% RSLogix 500 project HOT_WATER_SUPPLY.RSS, saved by version 8.30.00.16 %
PROJECT "BRAIN_1"    % processor: Bul.1763 MicroLogix 1100 Series B %

PROGRAM FILES
  LAD 2 "MAIN"  10 rungs
  LAD 3 "DIGI IN"  9 rungs  % Digital Inputs %
  LAD 4 "DIGI OUT"  6 rungs  % Digital Output %
  LAD 5 "ANG IN"  3 rungs  % Analog Inputs %
  LAD 6 "ANG OUT"  2 rungs  % Analog Output %
  LAD 7 "CONTROLS"  13 rungs  % Hand, Off, Auto Modes %
  LAD 9 "ALARMS"  21 rungs  % Alarms & Notification Control %
  LAD 10 "DISPLAY"  2 rungs

DATA FILES
  O0 OUTPUT  6 elements
  I1 INPUT  18 elements
  S2 STATUS  66 elements
  B3 BINARY  6 elements
  T4 TIMER  9 elements
  C5 COUNTER  1 elements
  R6 CONTROL  1 elements
  N7 INTEGER  10 elements
  F8 FLOAT  2 elements
  PD9 PID  1 elements

LADDER 2 "MAIN"
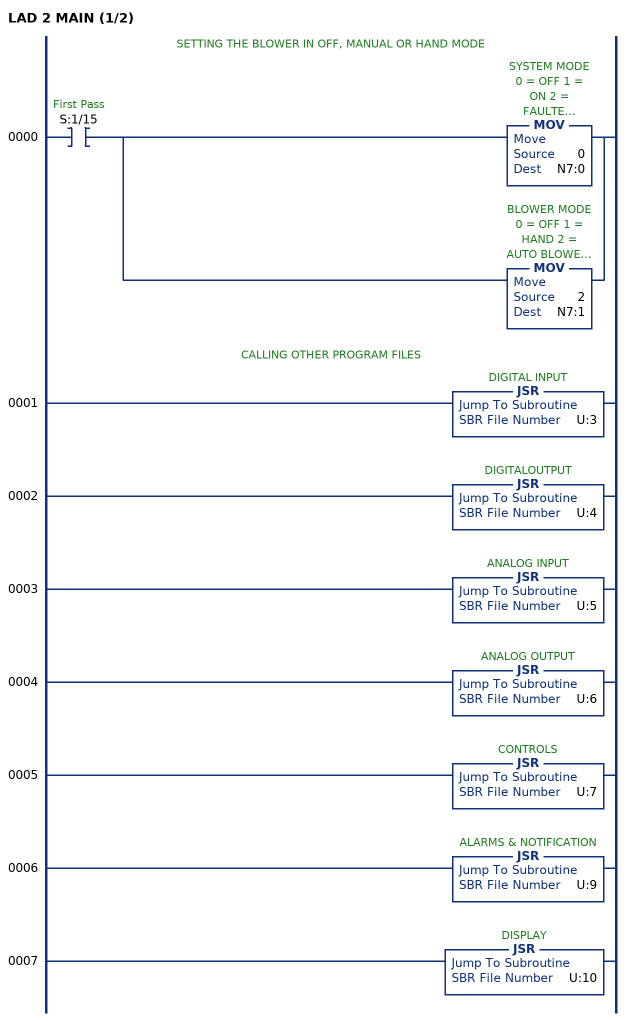
% Rung: 0 %
% SETTING THE BLOWER IN OFF, MANUAL OR HAND MODE %
SOR XIC S:1/15 BST MOV 0 N7:0 NXB MOV 2 N7:1 BND EOR
%   S:1/15  "First Pass" %
%   N7:0  SYSTEM_MODE  "SYSTEM MODE 0 = OFF 1 = ON 2 = FAULTED" %
%   N7:1  BLOWER_MODE  "BLOWER MODE 0 = OFF 1 = HAND 2 = AUTO" %
% Rung: 1 %
% CALLING OTHER PROGRAM FILES %
SOR JSR U:3 EOR
%   U:3  "DIGITAL INPUT" %
% Rung: 2 %
SOR JSR U:4 EOR
%   U:4  "DIGITALOUTPUT" %
% Rung: 3 %
SOR JSR U:5 EOR
%   U:5  "ANALOG INPUT" %
% Rung: 4 %
SOR JSR U:6 EOR
%   U:6  "ANALOG OUTPUT" %
% Rung: 5 %
SOR JSR U:7 EOR
%   U:7  "CONTROLS" %
% Rung: 6 %
SOR JSR U:9 EOR
%   U:9  "ALARMS & NOTIFICATION" %
% Rung: 7 %
SOR JSR U:10 EOR
%   U:10  "DISPLAY" %

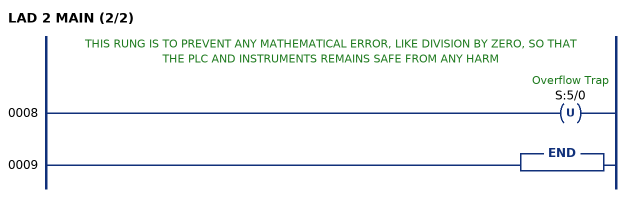
% Rung: 8 %
% THIS RUNG IS TO PREVENT ANY MATHEMATICAL ERROR, LIKE DIVISION BY ZERO, SO THAT THE PLC AND INSTRUMENTS REMAINS SAFE FROM ANY HARM %
SOR OTU S:5/0 EOR
%   S:5/0  "Overflow Trap" %
% Rung: 9 %
SOR END EOR

LADDER 3 "DIGI IN"    % Digital Inputs %
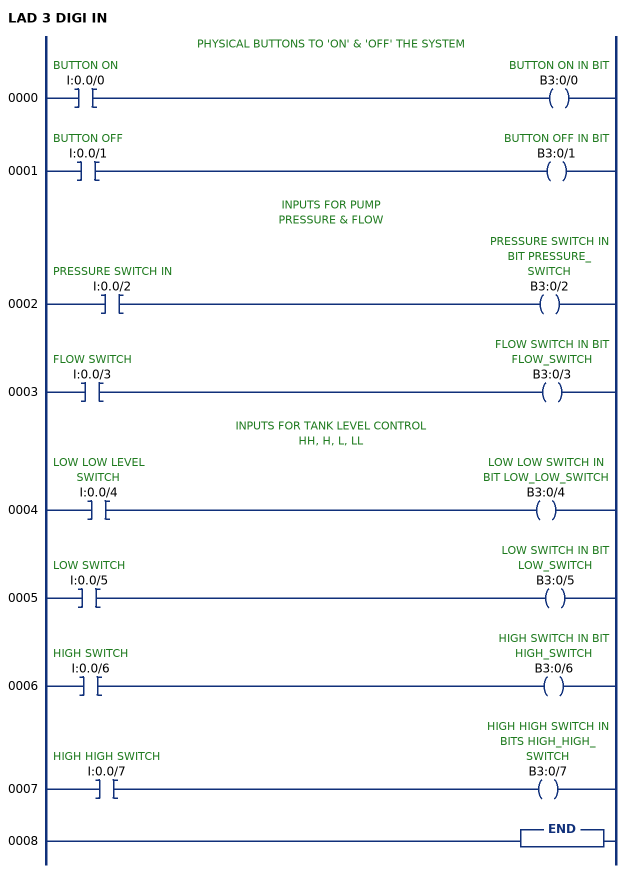
% Rung: 0 %
% PHYSICAL BUTTONS TO 'ON' & 'OFF' THE SYSTEM %
SOR XIC I:0.0/0 OTE B3:0/0 EOR
%   I:0.0/0  "BUTTON ON" %
%   B3:0/0  "BUTTON ON IN BIT" %
% Rung: 1 %
SOR XIC I:0.0/1 OTE B3:0/1 EOR
%   I:0.0/1  "BUTTON OFF" %
%   B3:0/1  "BUTTON OFF IN BIT" %
% Rung: 2 %
% INPUTS FOR PUMP
% PRESSURE & FLOW %
SOR XIC I:0.0/2 OTE B3:0/2 EOR
%   I:0.0/2  "PRESSURE SWITCH IN" %
%   B3:0/2  PRESSURE_SWITCH  "PRESSURE SWITCH IN BIT" %
% Rung: 3 %
SOR XIC I:0.0/3 OTE B3:0/3 EOR
%   I:0.0/3  "FLOW SWITCH" %
%   B3:0/3  FLOW_SWITCH  "FLOW SWITCH IN BIT" %
% Rung: 4 %
% INPUTS FOR TANK LEVEL CONTROL
% HH, H, L, LL %
SOR XIC I:0.0/4 OTE B3:0/4 EOR
%   I:0.0/4  "LOW LOW LEVEL SWITCH" %
%   B3:0/4  LOW_LOW_SWITCH  "LOW LOW SWITCH IN BIT" %
% Rung: 5 %
SOR XIC I:0.0/5 OTE B3:0/5 EOR
%   I:0.0/5  "LOW SWITCH" %
%   B3:0/5  LOW_SWITCH  "LOW SWITCH IN BIT" %
% Rung: 6 %
SOR XIC I:0.0/6 OTE B3:0/6 EOR
%   I:0.0/6  "HIGH SWITCH" %
%   B3:0/6  HIGH_SWITCH  "HIGH SWITCH IN BIT" %
% Rung: 7 %
SOR XIC I:0.0/7 OTE B3:0/7 EOR
%   I:0.0/7  "HIGH HIGH SWITCH" %
%   B3:0/7  HIGH_HIGH_SWITCH  "HIGH HIGH SWITCH IN BITS" %
% Rung: 8 %
SOR END EOR

LADDER 4 "DIGI OUT"    % Digital Output %
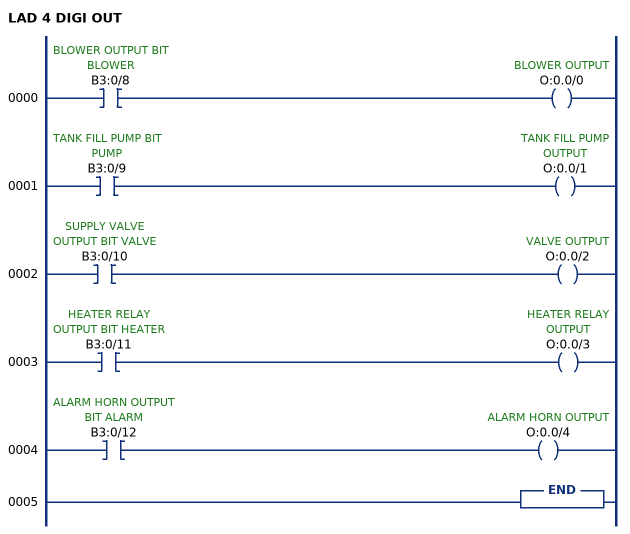
% Rung: 0 %
SOR XIC B3:0/8 OTE O:0.0/0 EOR
%   B3:0/8  BLOWER  "BLOWER OUTPUT BIT" %
%   O:0.0/0  "BLOWER OUTPUT" %
% Rung: 1 %
SOR XIC B3:0/9 OTE O:0.0/1 EOR
%   B3:0/9  PUMP  "TANK FILL PUMP BIT" %
%   O:0.0/1  "TANK FILL PUMP OUTPUT" %
% Rung: 2 %
SOR XIC B3:0/10 OTE O:0.0/2 EOR
%   B3:0/10  VALVE  "SUPPLY VALVE OUTPUT BIT" %
%   O:0.0/2  "VALVE OUTPUT" %
% Rung: 3 %
SOR XIC B3:0/11 OTE O:0.0/3 EOR
%   B3:0/11  HEATER  "HEATER RELAY OUTPUT BIT" %
%   O:0.0/3  "HEATER RELAY OUTPUT" %
% Rung: 4 %
SOR XIC B3:0/12 OTE O:0.0/4 EOR
%   B3:0/12  ALARM  "ALARM HORN OUTPUT BIT" %
%   O:0.0/4  "ALARM HORN OUTPUT" %
% Rung: 5 %
SOR END EOR

LADDER 5 "ANG IN"    % Analog Inputs %
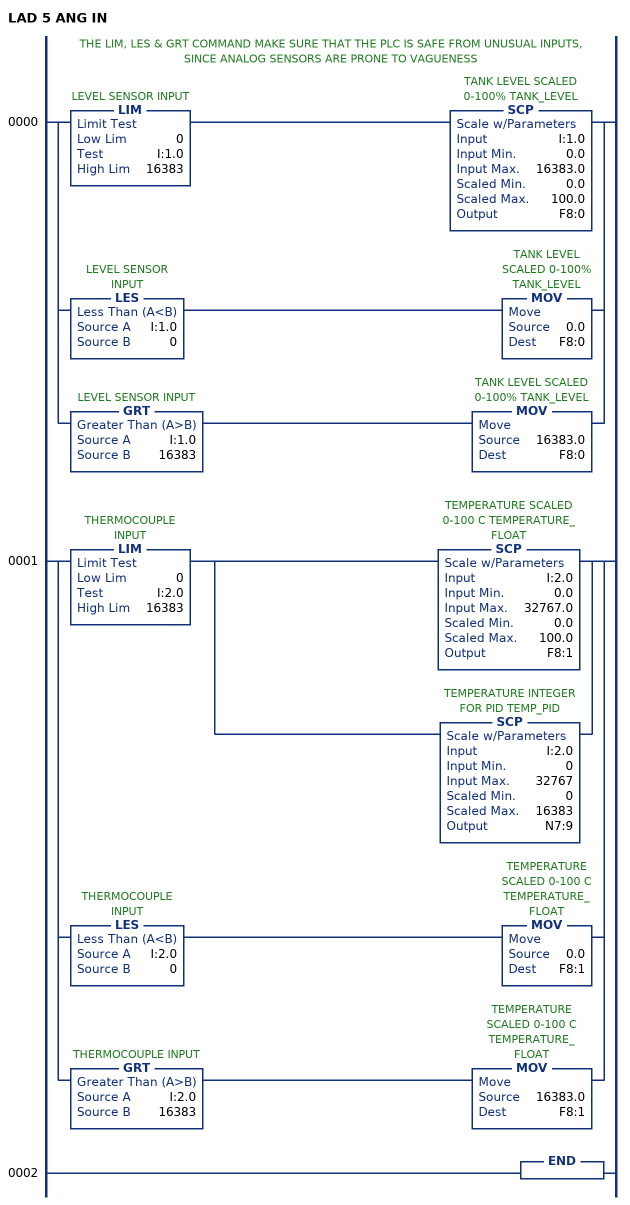
% Rung: 0 %
% THE LIM, LES & GRT COMMAND MAKE SURE THAT THE PLC IS SAFE FROM UNUSUAL INPUTS, SINCE ANALOG SENSORS ARE PRONE TO VAGUENESS %
SOR BST LIM 0 I:1.0 16383 SCP I:1.0 0.0 16383.0 0.0 100.0 F8:0 NXB BST LES I:1.0 0 MOV 0.0 F8:0 NXB GRT I:1.0 16383 MOV 16383.0 F8:0 BND BND EOR
%   I:1.0  "LEVEL SENSOR INPUT" %
%   F8:0  TANK_LEVEL  "TANK LEVEL SCALED 0-100%" %
% Rung: 1 %
SOR BST LIM 0 I:2.0 16383 BST SCP I:2.0 0.0 32767.0 0.0 100.0 F8:1 NXB SCP I:2.0 0 32767 0 16383 N7:9 BND NXB BST LES I:2.0 0 MOV 0.0 F8:1 NXB GRT I:2.0 16383 MOV 16383.0 F8:1 BND BND EOR
%   I:2.0  "THERMOCOUPLE INPUT" %
%   F8:1  TEMPERATURE_FLOAT  "TEMPERATURE SCALED 0-100 C" %
%   N7:9  TEMP_PID  "TEMPERATURE INTEGER FOR PID" %
% Rung: 2 %
SOR END EOR

LADDER 6 "ANG OUT"    % Analog Output %
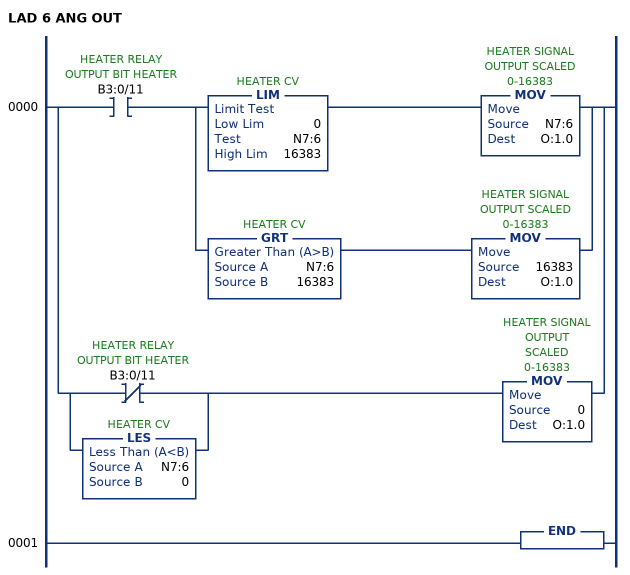
% Rung: 0 %
SOR BST XIC B3:0/11 BST LIM 0 N7:6 16383 MOV N7:6 O:1.0 NXB GRT N7:6 16383 MOV 16383 O:1.0 BND NXB BST XIO B3:0/11 NXB LES N7:6 0 BND MOV 0 O:1.0 BND EOR
%   B3:0/11  HEATER  "HEATER RELAY OUTPUT BIT" %
%   N7:6  "HEATER CV" %
%   O:1.0  "HEATER SIGNAL OUTPUT SCALED 0-16383" %
% Rung: 1 %
SOR END EOR

LADDER 7 "CONTROLS"    % Hand, Off, Auto Modes %
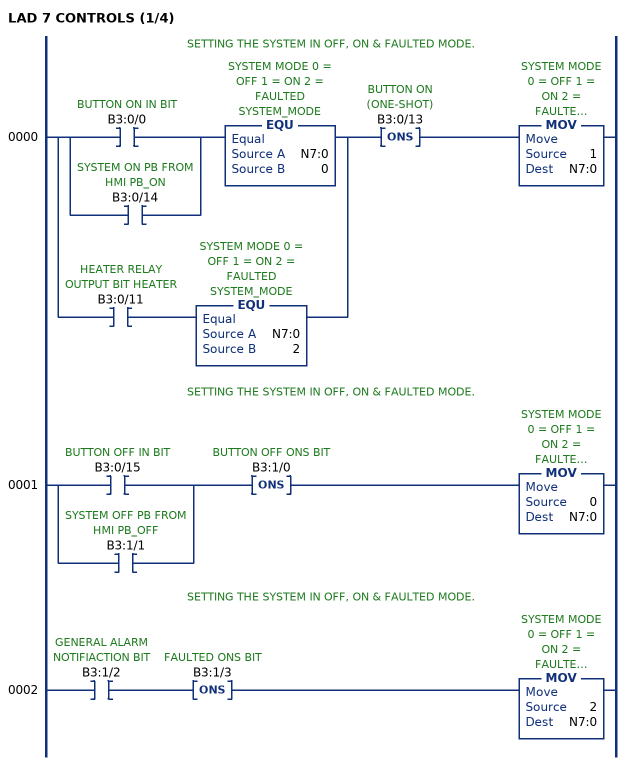
% Rung: 0 %
% SETTING THE SYSTEM IN OFF, ON & FAULTED MODE. %
SOR BST BST XIC B3:0/0 NXB XIC B3:0/14 BND EQU N7:0 0 NXB XIC B3:0/11 EQU N7:0 2 BND ONS B3:0/13 MOV 1 N7:0 EOR
%   B3:0/0  "BUTTON ON IN BIT" %
%   B3:0/14  PB_ON  "SYSTEM ON PB FROM HMI" %
%   N7:0  SYSTEM_MODE  "SYSTEM MODE 0 = OFF 1 = ON 2 = FAULTED" %
%   B3:0/11  HEATER  "HEATER RELAY OUTPUT BIT" %
%   B3:0/13  "BUTTON ON (ONE-SHOT)" %
% Rung: 1 %
% SETTING THE SYSTEM IN OFF, ON & FAULTED MODE. %
SOR BST XIC B3:0/15 NXB XIC B3:1/1 BND ONS B3:1/0 MOV 0 N7:0 EOR
%   B3:0/15  "BUTTON OFF IN BIT" %
%   B3:1/1  PB_OFF  "SYSTEM OFF PB FROM HMI" %
%   B3:1/0  "BUTTON OFF ONS BIT" %
%   N7:0  SYSTEM_MODE  "SYSTEM MODE 0 = OFF 1 = ON 2 = FAULTED" %
% Rung: 2 %
% SETTING THE SYSTEM IN OFF, ON & FAULTED MODE. %
SOR XIC B3:1/2 ONS B3:1/3 MOV 2 N7:0 EOR
%   B3:1/2  "GENERAL ALARM NOTIFIACTION BIT" %
%   B3:1/3  "FAULTED ONS BIT" %
%   N7:0  SYSTEM_MODE  "SYSTEM MODE 0 = OFF 1 = ON 2 = FAULTED" %

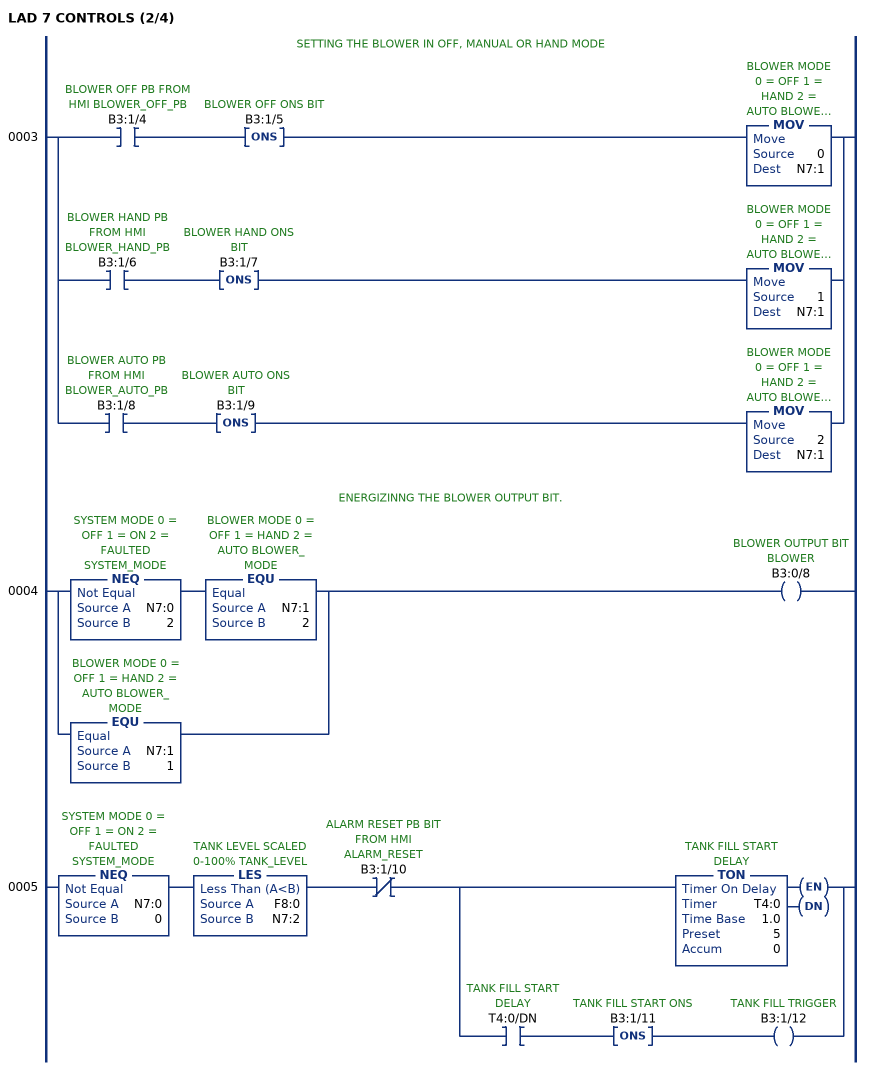
% Rung: 3 %
% SETTING THE BLOWER IN OFF, MANUAL OR HAND MODE %
SOR BST XIC B3:1/4 ONS B3:1/5 MOV 0 N7:1 NXB XIC B3:1/6 ONS B3:1/7 MOV 1 N7:1 NXB XIC B3:1/8 ONS B3:1/9 MOV 2 N7:1 BND EOR
%   B3:1/4  BLOWER_OFF_PB  "BLOWER OFF PB FROM HMI" %
%   B3:1/5  "BLOWER OFF ONS BIT" %
%   N7:1  BLOWER_MODE  "BLOWER MODE 0 = OFF 1 = HAND 2 = AUTO" %
%   B3:1/6  BLOWER_HAND_PB  "BLOWER HAND PB FROM HMI" %
%   B3:1/7  "BLOWER HAND ONS BIT" %
%   B3:1/8  BLOWER_AUTO_PB  "BLOWER AUTO PB FROM HMI" %
%   B3:1/9  "BLOWER AUTO ONS BIT" %
% Rung: 4 %
% ENERGIZINNG THE BLOWER OUTPUT BIT. %
SOR BST NEQ N7:0 2 EQU N7:1 2 NXB EQU N7:1 1 BND OTE B3:0/8 EOR
%   N7:0  SYSTEM_MODE  "SYSTEM MODE 0 = OFF 1 = ON 2 = FAULTED" %
%   N7:1  BLOWER_MODE  "BLOWER MODE 0 = OFF 1 = HAND 2 = AUTO" %
%   B3:0/8  BLOWER  "BLOWER OUTPUT BIT" %
% Rung: 5 %
SOR NEQ N7:0 0 LES F8:0 N7:2 XIO B3:1/10 BST TON T4:0 1.0 5 0 NXB XIC T4:0/DN ONS B3:1/11 OTE B3:1/12 BND EOR
%   N7:0  SYSTEM_MODE  "SYSTEM MODE 0 = OFF 1 = ON 2 = FAULTED" %
%   F8:0  TANK_LEVEL  "TANK LEVEL SCALED 0-100%" %
%   N7:2  TANK_LOW_SP  "TANK LOW SETPOINT" %
%   B3:1/10  ALARM_RESET  "ALARM RESET PB BIT FROM HMI" %
%   T4:0  "TANK FILL START DELAY" %
%   B3:1/11  "TANK FILL START ONS" %
%   B3:1/12  "TANK FILL TRIGGER" %

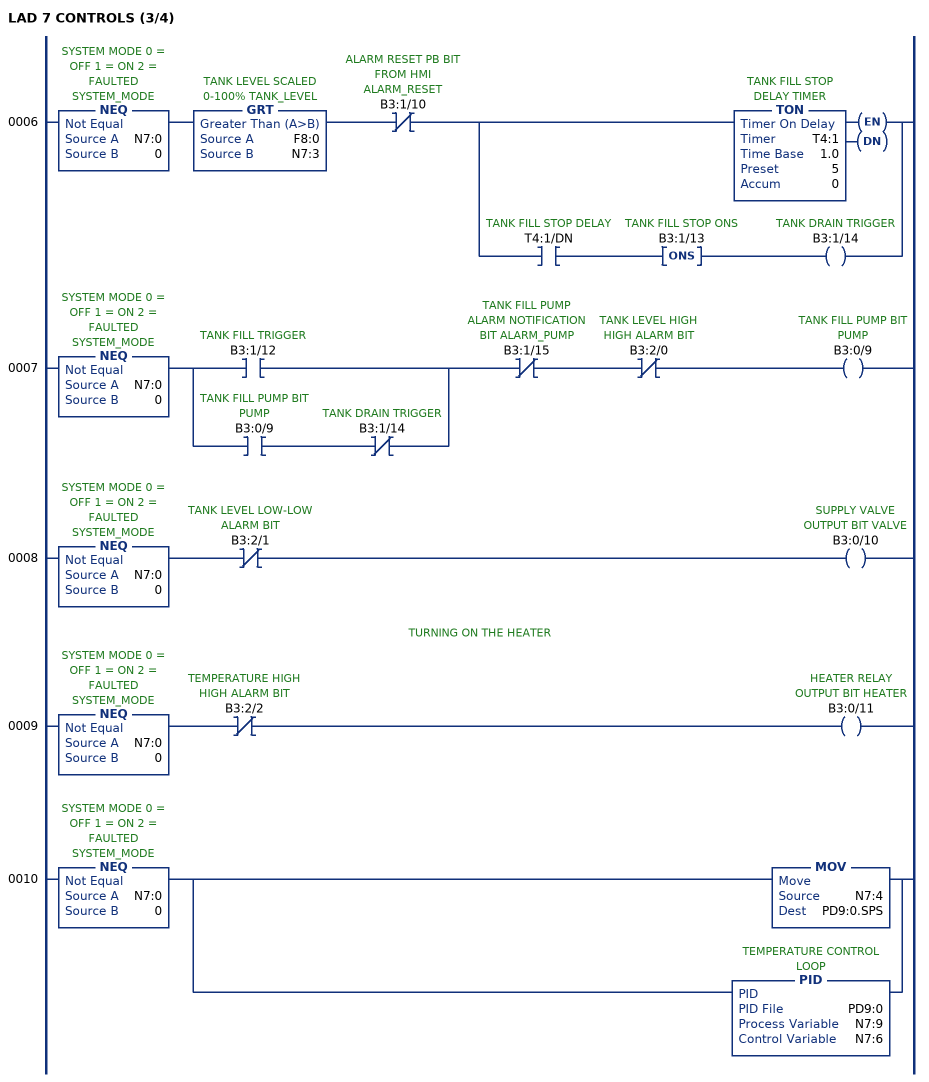
% Rung: 6 %
SOR NEQ N7:0 0 GRT F8:0 N7:3 XIO B3:1/10 BST TON T4:1 1.0 5 0 NXB XIC T4:1/DN ONS B3:1/13 OTE B3:1/14 BND EOR
%   N7:0  SYSTEM_MODE  "SYSTEM MODE 0 = OFF 1 = ON 2 = FAULTED" %
%   F8:0  TANK_LEVEL  "TANK LEVEL SCALED 0-100%" %
%   N7:3  TANK_HIGH_SP  "TANK HIGH SETPOINT" %
%   B3:1/10  ALARM_RESET  "ALARM RESET PB BIT FROM HMI" %
%   T4:1  "TANK FILL STOP DELAY TIMER" %
%   T4:1/DN  "TANK FILL STOP DELAY" %
%   B3:1/13  "TANK FILL STOP ONS" %
%   B3:1/14  "TANK DRAIN TRIGGER" %
% Rung: 7 %
SOR NEQ N7:0 0 BST XIC B3:1/12 NXB XIC B3:0/9 XIO B3:1/14 BND XIO B3:1/15 XIO B3:2/0 OTE B3:0/9 EOR
%   N7:0  SYSTEM_MODE  "SYSTEM MODE 0 = OFF 1 = ON 2 = FAULTED" %
%   B3:1/12  "TANK FILL TRIGGER" %
%   B3:0/9  PUMP  "TANK FILL PUMP BIT" %
%   B3:1/14  "TANK DRAIN TRIGGER" %
%   B3:1/15  ALARM_PUMP  "TANK FILL PUMP ALARM NOTIFICATION BIT" %
%   B3:2/0  "TANK LEVEL HIGH HIGH ALARM BIT" %
% Rung: 8 %
SOR NEQ N7:0 0 XIO B3:2/1 OTE B3:0/10 EOR
%   N7:0  SYSTEM_MODE  "SYSTEM MODE 0 = OFF 1 = ON 2 = FAULTED" %
%   B3:2/1  "TANK LEVEL LOW-LOW ALARM BIT" %
%   B3:0/10  VALVE  "SUPPLY VALVE OUTPUT BIT" %
% Rung: 9 %
% TURNING ON THE HEATER %
SOR NEQ N7:0 0 XIO B3:2/2 OTE B3:0/11 EOR
%   N7:0  SYSTEM_MODE  "SYSTEM MODE 0 = OFF 1 = ON 2 = FAULTED" %
%   B3:2/2  "TEMPERATURE HIGH HIGH ALARM BIT" %
%   B3:0/11  HEATER  "HEATER RELAY OUTPUT BIT" %
% Rung: 10 %
SOR NEQ N7:0 0 BST MOV N7:4 PD9:0.SPS NXB PID PD9:0 N7:9 N7:6 BND EOR
%   N7:0  SYSTEM_MODE  "SYSTEM MODE 0 = OFF 1 = ON 2 = FAULTED" %
%   N7:4  TEMP_SETPOINT  "TEMP SETPOINT" %
%   PD9:0  "TEMPERATURE CONTROL LOOP" %
%   N7:9  TEMP_PID  "TEMPERATURE INTEGER FOR PID" %
%   N7:6  "HEATER CV" %

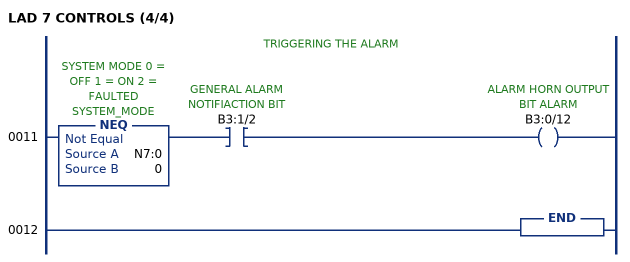
% Rung: 11 %
% TRIGGERING THE ALARM %
SOR NEQ N7:0 0 XIC B3:1/2 OTE B3:0/12 EOR
%   N7:0  SYSTEM_MODE  "SYSTEM MODE 0 = OFF 1 = ON 2 = FAULTED" %
%   B3:1/2  "GENERAL ALARM NOTIFIACTION BIT" %
%   B3:0/12  ALARM  "ALARM HORN OUTPUT BIT" %
% Rung: 12 %
SOR END EOR

LADDER 9 "ALARMS"    % Alarms & Notification Control %
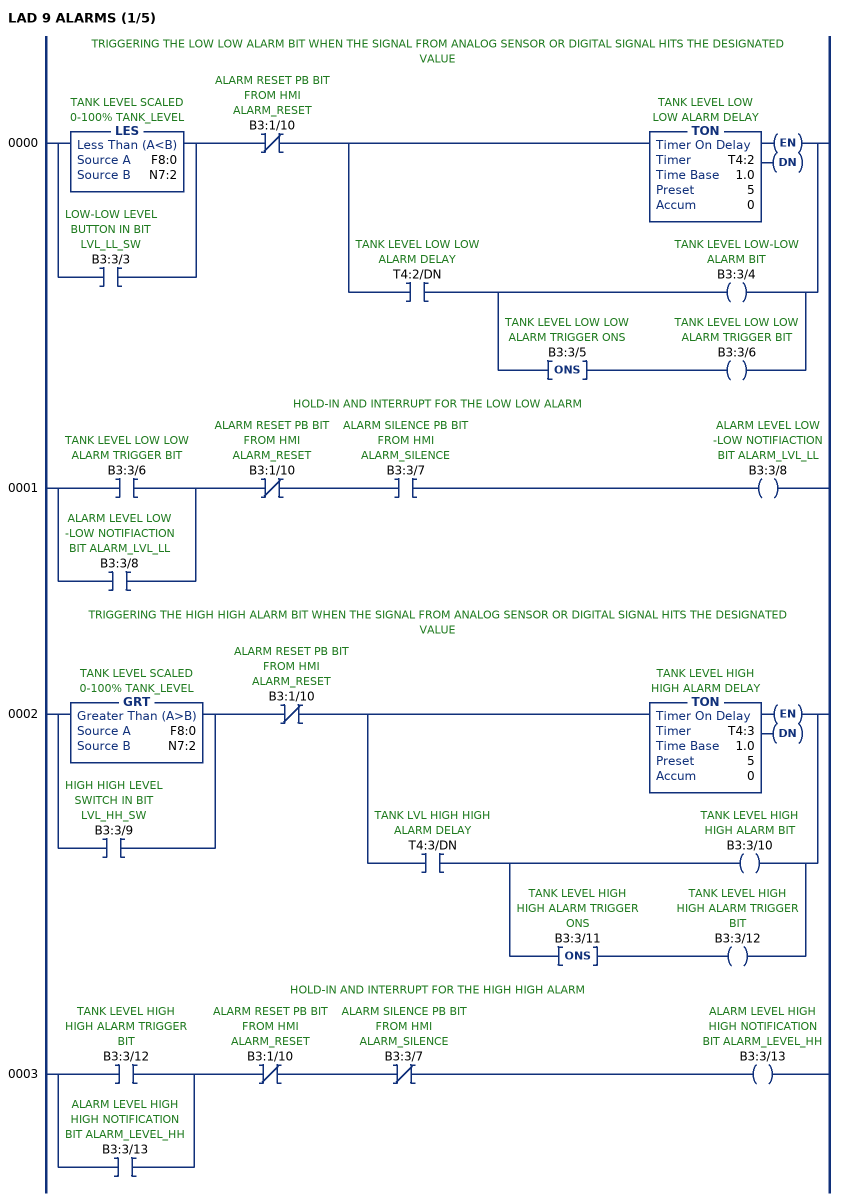
% Rung: 0 %
% TRIGGERING THE LOW LOW ALARM BIT WHEN THE SIGNAL FROM ANALOG SENSOR OR DIGITAL SIGNAL HITS THE DESIGNATED VALUE %
SOR BST LES F8:0 N7:2 NXB XIC B3:3/3 BND XIO B3:1/10 BST TON T4:2 1.0 5 0 NXB XIC T4:2/DN BST OTE B3:3/4 NXB ONS B3:3/5 OTE B3:3/6 BND BND EOR
%   F8:0  TANK_LEVEL  "TANK LEVEL SCALED 0-100%" %
%   N7:2  TANK_LOW_SP  "TANK LOW SETPOINT" %
%   B3:3/3  LVL_LL_SW  "LOW-LOW LEVEL BUTTON IN BIT" %
%   B3:1/10  ALARM_RESET  "ALARM RESET PB BIT FROM HMI" %
%   T4:2  "TANK LEVEL LOW LOW ALARM DELAY" %
%   B3:3/4  "TANK LEVEL LOW-LOW ALARM BIT" %
%   B3:3/5  "TANK LEVEL LOW LOW ALARM TRIGGER ONS" %
%   B3:3/6  "TANK LEVEL LOW LOW ALARM TRIGGER BIT" %
% Rung: 1 %
% HOLD-IN AND INTERRUPT FOR THE LOW LOW ALARM %
SOR BST XIC B3:3/6 NXB XIC B3:3/8 BND XIO B3:1/10 XIC B3:3/7 OTE B3:3/8 EOR
%   B3:3/6  "TANK LEVEL LOW LOW ALARM TRIGGER BIT" %
%   B3:3/8  ALARM_LVL_LL  "ALARM LEVEL LOW -LOW NOTIFIACTION BIT" %
%   B3:1/10  ALARM_RESET  "ALARM RESET PB BIT FROM HMI" %
%   B3:3/7  ALARM_SILENCE  "ALARM SILENCE PB BIT FROM HMI" %
% Rung: 2 %
% TRIGGERING THE HIGH HIGH ALARM BIT WHEN THE SIGNAL FROM ANALOG SENSOR OR DIGITAL SIGNAL HITS THE DESIGNATED VALUE %
SOR BST GRT F8:0 N7:2 NXB XIC B3:3/9 BND XIO B3:1/10 BST TON T4:3 1.0 5 0 NXB XIC T4:3/DN BST OTE B3:3/10 NXB ONS B3:3/11 OTE B3:3/12 BND BND EOR
%   F8:0  TANK_LEVEL  "TANK LEVEL SCALED 0-100%" %
%   N7:2  TANK_LOW_SP  "TANK LOW SETPOINT" %
%   B3:3/9  LVL_HH_SW  "HIGH HIGH LEVEL SWITCH IN BIT" %
%   B3:1/10  ALARM_RESET  "ALARM RESET PB BIT FROM HMI" %
%   T4:3  "TANK LEVEL HIGH HIGH ALARM DELAY" %
%   T4:3/DN  "TANK LVL HIGH HIGH ALARM DELAY" %
%   B3:3/10  "TANK LEVEL HIGH HIGH ALARM BIT" %
%   B3:3/11  "TANK LEVEL HIGH HIGH ALARM TRIGGER ONS" %
%   B3:3/12  "TANK LEVEL HIGH HIGH ALARM TRIGGER BIT" %
% Rung: 3 %
% HOLD-IN AND INTERRUPT FOR THE HIGH HIGH ALARM %
SOR BST XIC B3:3/12 NXB XIC B3:3/13 BND XIO B3:1/10 XIO B3:3/7 OTE B3:3/13 EOR
%   B3:3/12  "TANK LEVEL HIGH HIGH ALARM TRIGGER BIT" %
%   B3:3/13  ALARM_LEVEL_HH  "ALARM LEVEL HIGH HIGH NOTIFICATION BIT" %
%   B3:1/10  ALARM_RESET  "ALARM RESET PB BIT FROM HMI" %
%   B3:3/7  ALARM_SILENCE  "ALARM SILENCE PB BIT FROM HMI" %

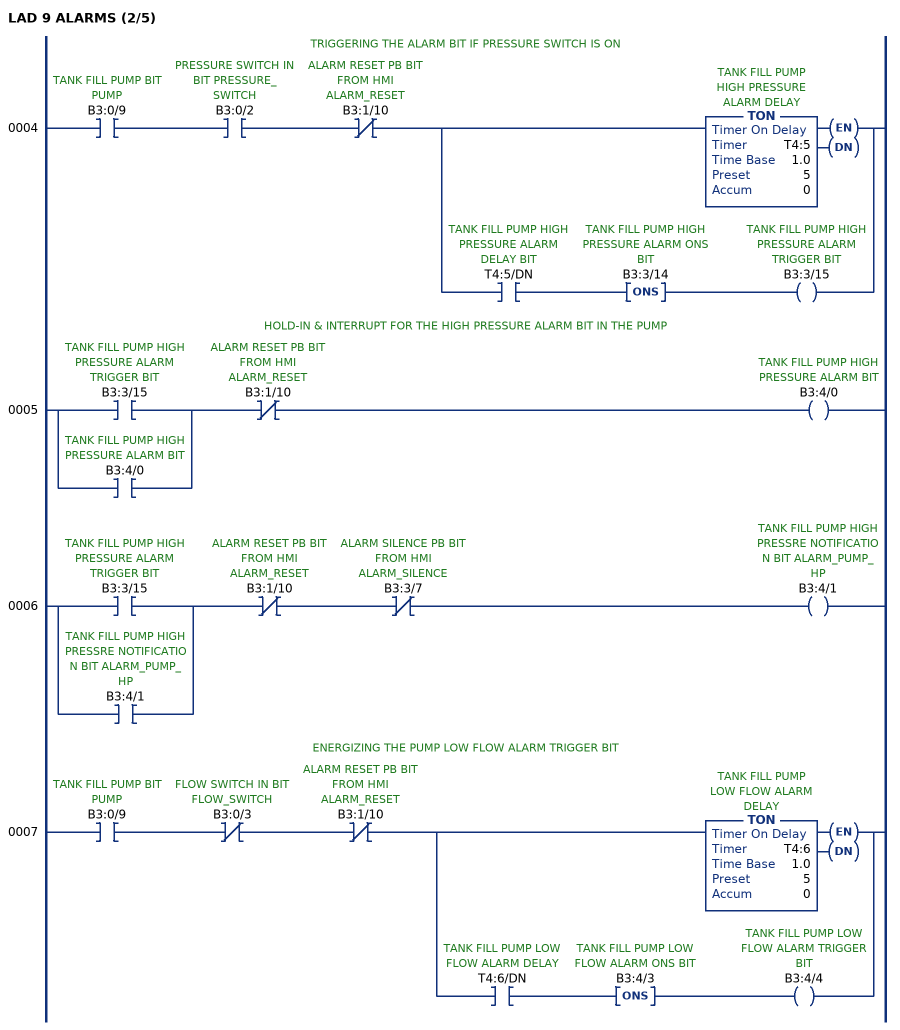
% Rung: 4 %
% TRIGGERING THE ALARM BIT IF PRESSURE SWITCH IS ON %
SOR XIC B3:0/9 XIC B3:0/2 XIO B3:1/10 BST TON T4:5 1.0 5 0 NXB XIC T4:5/DN ONS B3:3/14 OTE B3:3/15 BND EOR
%   B3:0/9  PUMP  "TANK FILL PUMP BIT" %
%   B3:0/2  PRESSURE_SWITCH  "PRESSURE SWITCH IN BIT" %
%   B3:1/10  ALARM_RESET  "ALARM RESET PB BIT FROM HMI" %
%   T4:5  "TANK FILL PUMP HIGH PRESSURE ALARM DELAY" %
%   T4:5/DN  "TANK FILL PUMP HIGH PRESSURE ALARM DELAY BIT" %
%   B3:3/14  "TANK FILL PUMP HIGH PRESSURE ALARM ONS BIT" %
%   B3:3/15  "TANK FILL PUMP HIGH PRESSURE ALARM TRIGGER BIT" %
% Rung: 5 %
% HOLD-IN & INTERRUPT FOR THE HIGH PRESSURE ALARM BIT IN THE PUMP %
SOR BST XIC B3:3/15 NXB XIC B3:4/0 BND XIO B3:1/10 OTE B3:4/0 EOR
%   B3:3/15  "TANK FILL PUMP HIGH PRESSURE ALARM TRIGGER BIT" %
%   B3:4/0  "TANK FILL PUMP HIGH PRESSURE ALARM BIT" %
%   B3:1/10  ALARM_RESET  "ALARM RESET PB BIT FROM HMI" %
% Rung: 6 %
SOR BST XIC B3:3/15 NXB XIC B3:4/1 BND XIO B3:1/10 XIO B3:3/7 OTE B3:4/1 EOR
%   B3:3/15  "TANK FILL PUMP HIGH PRESSURE ALARM TRIGGER BIT" %
%   B3:4/1  ALARM_PUMP_HP  "TANK FILL PUMP HIGH PRESSRE NOTIFICATION BIT" %
%   B3:1/10  ALARM_RESET  "ALARM RESET PB BIT FROM HMI" %
%   B3:3/7  ALARM_SILENCE  "ALARM SILENCE PB BIT FROM HMI" %
% Rung: 7 %
% ENERGIZING THE PUMP LOW FLOW ALARM TRIGGER BIT %
SOR XIC B3:0/9 XIO B3:0/3 XIO B3:1/10 BST TON T4:6 1.0 5 0 NXB XIC T4:6/DN ONS B3:4/3 OTE B3:4/4 BND EOR
%   B3:0/9  PUMP  "TANK FILL PUMP BIT" %
%   B3:0/3  FLOW_SWITCH  "FLOW SWITCH IN BIT" %
%   B3:1/10  ALARM_RESET  "ALARM RESET PB BIT FROM HMI" %
%   T4:6  "TANK FILL PUMP LOW FLOW ALARM DELAY" %
%   T4:6/DN  "TANK FILL PUMP LOW FLOW ALARM DELAY" %
%   B3:4/3  "TANK FILL PUMP LOW FLOW ALARM ONS BIT" %
%   B3:4/4  "TANK FILL PUMP LOW FLOW ALARM TRIGGER BIT" %

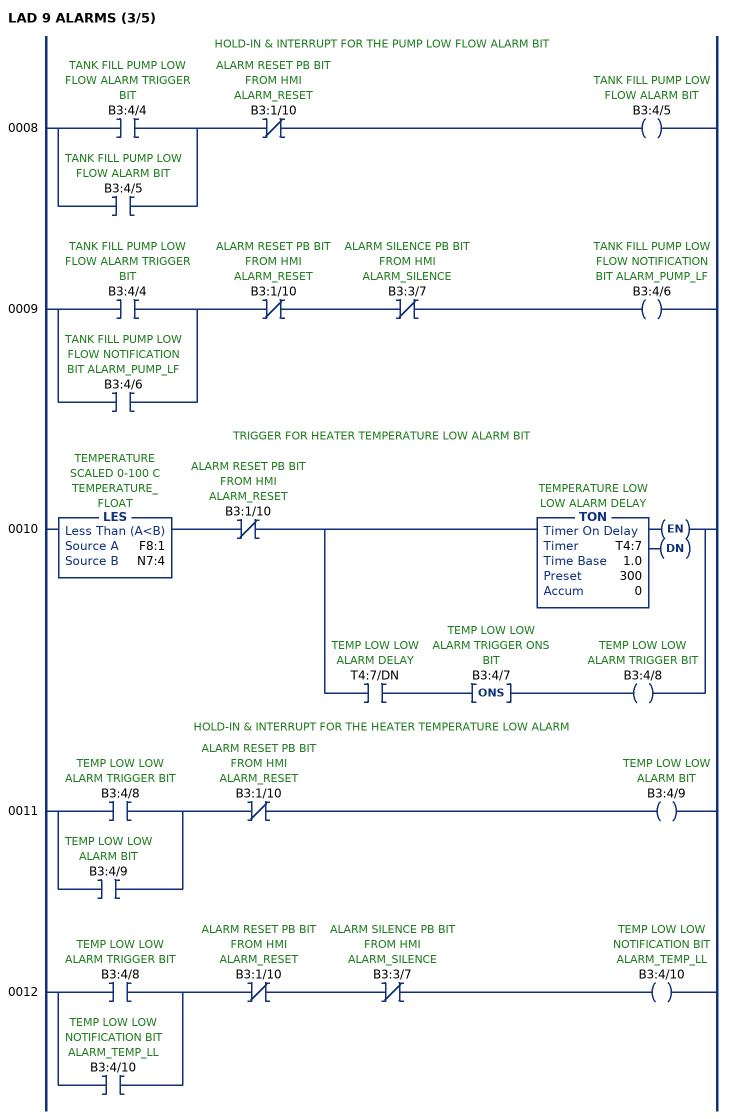
% Rung: 8 %
% HOLD-IN & INTERRUPT FOR THE PUMP LOW FLOW ALARM BIT %
SOR BST XIC B3:4/4 NXB XIC B3:4/5 BND XIO B3:1/10 OTE B3:4/5 EOR
%   B3:4/4  "TANK FILL PUMP LOW FLOW ALARM TRIGGER BIT" %
%   B3:4/5  "TANK FILL PUMP LOW FLOW ALARM BIT" %
%   B3:1/10  ALARM_RESET  "ALARM RESET PB BIT FROM HMI" %
% Rung: 9 %
SOR BST XIC B3:4/4 NXB XIC B3:4/6 BND XIO B3:1/10 XIO B3:3/7 OTE B3:4/6 EOR
%   B3:4/4  "TANK FILL PUMP LOW FLOW ALARM TRIGGER BIT" %
%   B3:4/6  ALARM_PUMP_LF  "TANK FILL PUMP LOW FLOW NOTIFICATION BIT" %
%   B3:1/10  ALARM_RESET  "ALARM RESET PB BIT FROM HMI" %
%   B3:3/7  ALARM_SILENCE  "ALARM SILENCE PB BIT FROM HMI" %
% Rung: 10 %
% TRIGGER FOR HEATER TEMPERATURE LOW ALARM BIT %
SOR LES F8:1 N7:4 XIO B3:1/10 BST TON T4:7 1.0 300 0 NXB XIC T4:7/DN ONS B3:4/7 OTE B3:4/8 BND EOR
%   F8:1  TEMPERATURE_FLOAT  "TEMPERATURE SCALED 0-100 C" %
%   N7:4  TEMP_SETPOINT  "TEMP SETPOINT" %
%   B3:1/10  ALARM_RESET  "ALARM RESET PB BIT FROM HMI" %
%   T4:7  "TEMPERATURE LOW LOW ALARM DELAY" %
%   T4:7/DN  "TEMP LOW LOW ALARM DELAY" %
%   B3:4/7  "TEMP LOW LOW ALARM TRIGGER ONS BIT" %
%   B3:4/8  "TEMP LOW LOW ALARM TRIGGER BIT" %
% Rung: 11 %
% HOLD-IN & INTERRUPT FOR THE HEATER TEMPERATURE LOW ALARM %
SOR BST XIC B3:4/8 NXB XIC B3:4/9 BND XIO B3:1/10 OTE B3:4/9 EOR
%   B3:4/8  "TEMP LOW LOW ALARM TRIGGER BIT" %
%   B3:4/9  "TEMP LOW LOW ALARM BIT" %
%   B3:1/10  ALARM_RESET  "ALARM RESET PB BIT FROM HMI" %
% Rung: 12 %
SOR BST XIC B3:4/8 NXB XIC B3:4/10 BND XIO B3:1/10 XIO B3:3/7 OTE B3:4/10 EOR
%   B3:4/8  "TEMP LOW LOW ALARM TRIGGER BIT" %
%   B3:4/10  ALARM_TEMP_LL  "TEMP LOW LOW NOTIFICATION BIT" %
%   B3:1/10  ALARM_RESET  "ALARM RESET PB BIT FROM HMI" %
%   B3:3/7  ALARM_SILENCE  "ALARM SILENCE PB BIT FROM HMI" %

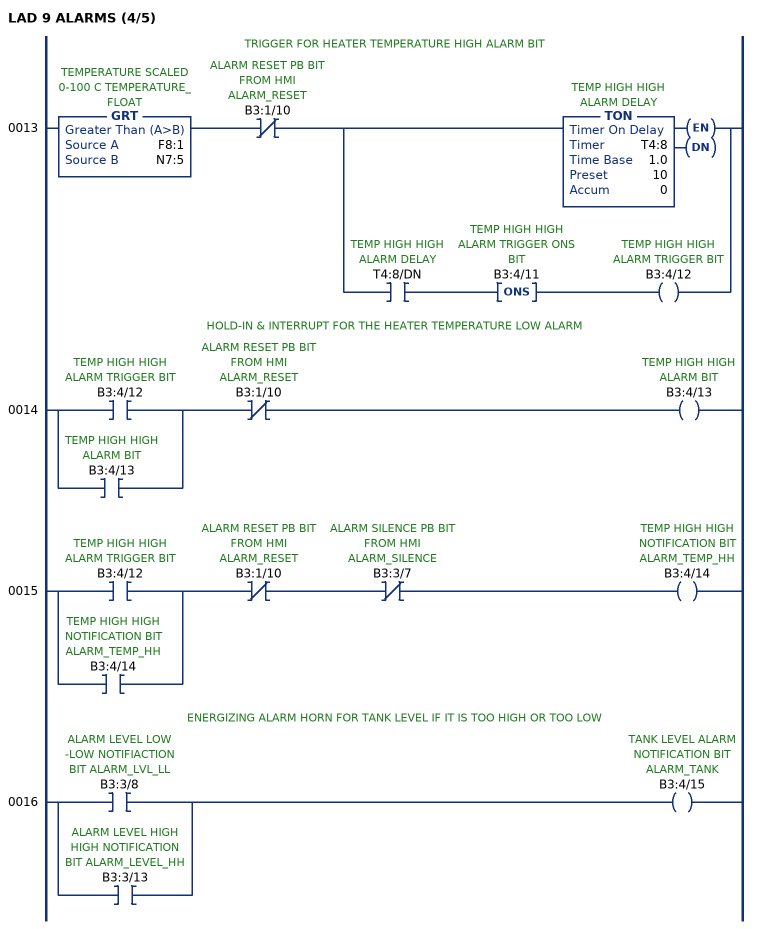
% Rung: 13 %
% TRIGGER FOR HEATER TEMPERATURE HIGH ALARM BIT %
SOR GRT F8:1 N7:5 XIO B3:1/10 BST TON T4:8 1.0 10 0 NXB XIC T4:8/DN ONS B3:4/11 OTE B3:4/12 BND EOR
%   F8:1  TEMPERATURE_FLOAT  "TEMPERATURE SCALED 0-100 C" %
%   N7:5  TEMP_HH_SETPOINT  "TEMP HIGH HIGH SETPOINT" %
%   B3:1/10  ALARM_RESET  "ALARM RESET PB BIT FROM HMI" %
%   T4:8  "TEMP HIGH HIGH ALARM DELAY" %
%   T4:8/DN  "TEMP HIGH HIGH ALARM DELAY" %
%   B3:4/11  "TEMP HIGH HIGH ALARM TRIGGER ONS BIT" %
%   B3:4/12  "TEMP HIGH HIGH ALARM TRIGGER BIT" %
% Rung: 14 %
% HOLD-IN & INTERRUPT FOR THE HEATER TEMPERATURE LOW ALARM %
SOR BST XIC B3:4/12 NXB XIC B3:4/13 BND XIO B3:1/10 OTE B3:4/13 EOR
%   B3:4/12  "TEMP HIGH HIGH ALARM TRIGGER BIT" %
%   B3:4/13  "TEMP HIGH HIGH ALARM BIT" %
%   B3:1/10  ALARM_RESET  "ALARM RESET PB BIT FROM HMI" %
% Rung: 15 %
SOR BST XIC B3:4/12 NXB XIC B3:4/14 BND XIO B3:1/10 XIO B3:3/7 OTE B3:4/14 EOR
%   B3:4/12  "TEMP HIGH HIGH ALARM TRIGGER BIT" %
%   B3:4/14  ALARM_TEMP_HH  "TEMP HIGH HIGH NOTIFICATION BIT" %
%   B3:1/10  ALARM_RESET  "ALARM RESET PB BIT FROM HMI" %
%   B3:3/7  ALARM_SILENCE  "ALARM SILENCE PB BIT FROM HMI" %
% Rung: 16 %
% ENERGIZING ALARM HORN FOR TANK LEVEL IF IT IS TOO HIGH OR TOO LOW %
SOR BST XIC B3:3/8 NXB XIC B3:3/13 BND OTE B3:4/15 EOR
%   B3:3/8  ALARM_LVL_LL  "ALARM LEVEL LOW -LOW NOTIFIACTION BIT" %
%   B3:3/13  ALARM_LEVEL_HH  "ALARM LEVEL HIGH HIGH NOTIFICATION BIT" %
%   B3:4/15  ALARM_TANK  "TANK LEVEL ALARM NOTIFICATION BIT" %

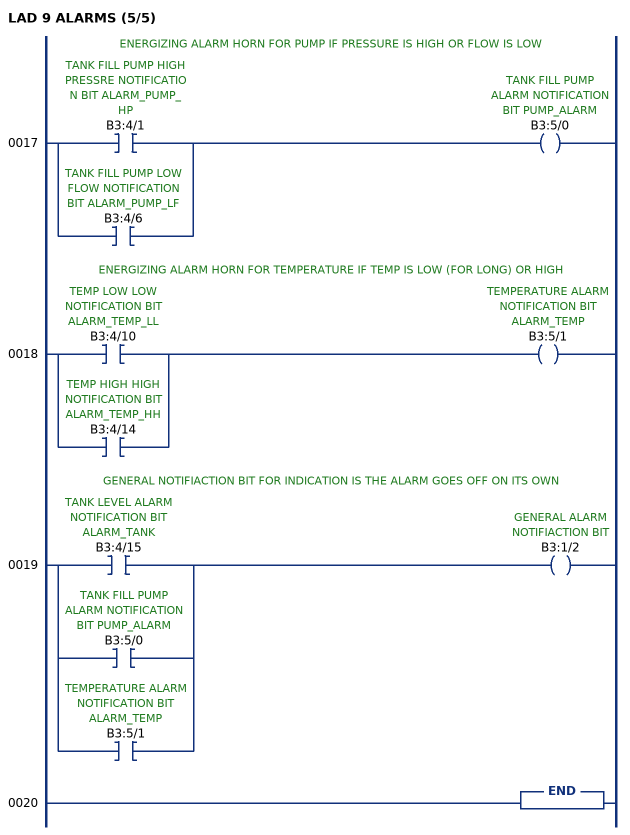
% Rung: 17 %
% ENERGIZING ALARM HORN FOR PUMP IF PRESSURE IS HIGH OR FLOW IS LOW %
SOR BST XIC B3:4/1 NXB XIC B3:4/6 BND OTE B3:5/0 EOR
%   B3:4/1  ALARM_PUMP_HP  "TANK FILL PUMP HIGH PRESSRE NOTIFICATION BIT" %
%   B3:4/6  ALARM_PUMP_LF  "TANK FILL PUMP LOW FLOW NOTIFICATION BIT" %
%   B3:5/0  PUMP_ALARM  "TANK FILL PUMP ALARM NOTIFICATION BIT" %
% Rung: 18 %
% ENERGIZING ALARM HORN FOR TEMPERATURE IF TEMP IS LOW (FOR LONG) OR HIGH %
SOR BST XIC B3:4/10 NXB XIC B3:4/14 BND OTE B3:5/1 EOR
%   B3:4/10  ALARM_TEMP_LL  "TEMP LOW LOW NOTIFICATION BIT" %
%   B3:4/14  ALARM_TEMP_HH  "TEMP HIGH HIGH NOTIFICATION BIT" %
%   B3:5/1  ALARM_TEMP  "TEMPERATURE ALARM NOTIFICATION BIT" %
% Rung: 19 %
% GENERAL NOTIFIACTION BIT FOR INDICATION IS THE ALARM GOES OFF ON ITS OWN %
SOR BST XIC B3:4/15 NXB XIC B3:5/0 NXB XIC B3:5/1 BND OTE B3:1/2 EOR
%   B3:4/15  ALARM_TANK  "TANK LEVEL ALARM NOTIFICATION BIT" %
%   B3:5/0  PUMP_ALARM  "TANK FILL PUMP ALARM NOTIFICATION BIT" %
%   B3:5/1  ALARM_TEMP  "TEMPERATURE ALARM NOTIFICATION BIT" %
%   B3:1/2  "GENERAL ALARM NOTIFIACTION BIT" %
% Rung: 20 %
SOR END EOR

LADDER 10 "DISPLAY"
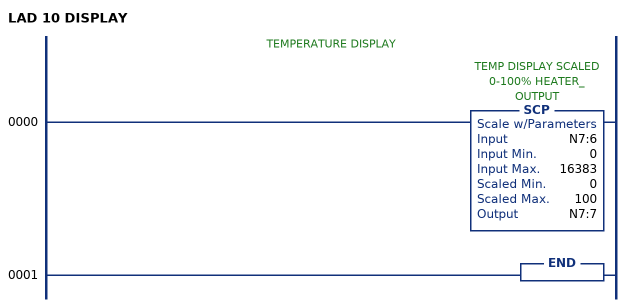
% Rung: 0 %
% TEMPERATURE DISPLAY %
SOR SCP N7:6 0 16383 0 100 N7:7 EOR
%   N7:6  "HEATER CV" %
%   N7:7  HEATER_OUTPUT  "TEMP DISPLAY SCALED 0-100%" %
% Rung: 1 %
SOR END EOR

OTHER DOCUMENTED ADDRESSES
  B3:4/2  "FLOW SWITCH IN BIT"
  B4:1/5  "BLOWER OFF ONS BIT"
  B4:1/7  "BLOWER HAND ONS BIT"
  B4:1/9  "BLOWER AUTO ONS BIT"
  EQU  
  I:1.0/0  "LEVEL SENSOR INPUT"
  I:2.0/0  "THERMOCOUPLE INPUT"
  MOV  
  O:1.0/0  "HEATER SIGNAL OUTPUT SCALED 0-16383"
  PD9:0.2  "TEMPERATURE CONTROL LOOP"
  PFILE:8  "Process Controls"
  PID  
  U:8  "COTROLS"

COMMENTS NOT ATTACHED TO A CURRENT RUNG
  O:1.0/0: IF THE HEATER IS 'ON' AND PASSES THE LES OR GRT COMMAND THEN PERFORM MOV COMMAND
    IF THE HEATER IS 'OFF' OR LES COMMAND IS MET MOVCOMMAND IS EXECUTED -- 0 TO OUTPUT
  T4:0: CONTROL TO FILL THE TANK
  T4:1: CONTROLS TO DRAIN THE TANK
  PD9:0.2: CONTROLLING THE TEMPERATURE WITH PID AS PER THE DESIGNATED SETPOINT

REVISION NOTES
  0: PID SETUP---FLOAT PROBLEM
     INTEGER LINED UP CHECK IF IT IS OKAY

DATA TABLE (non-zero values as saved)
DATA T4
% .PRE .ACC %
% T4:0 % 5 0
% T4:1 % 5 0
% T4:2 % 5 0
% T4:3 % 5 0
% T4:5 % 5 0
% T4:6 % 5 0
% T4:7 % 300 0
% T4:8 % 10 0
